KUKA KRL data list: $config.dat

&ACCESS RV$4
DEFDAT $CONFIG

ENDDAT
